FUNCTION_BLOCK TEST2
VAR_INPUT
END_VAR
VAR_OUTPUT
END_VAR
VAR
END_VAR

END_FUNCTION_BLOCK

(* stored: Version 1.1.0.1, ProductVersion 3.1.4024.14
   POU TEST2: Id {9d48b9b3-5efd-469d-8dc8-c79a998fc515}, SpecialFunc None *)
